{attribute 'GeneratedUsingTerminal: EL1512-0000-0016'}
{attribute addProperty BoxType "EL1512-0000-0016"}
{attribute addProperty Id "Set_counterAT %Q*BOOL1Inhibit_counterAT %Q*BOOL1Set_counter_valueAT %Q*UDINT4"}
{attribute addProperty CRC "2001350844"}
{attribute addProperty Size "6"}
TYPE CNT_Outputs_Channel_774A30BC :
STRUCT
	{attribute addProperty Name "Set_counter"}
	Set_counter AT %Q* : BOOL;
	{attribute addProperty Name "Inhibit_counter"}
	Inhibit_counter AT %Q* : BOOL;
	{attribute addProperty Name "Set_counter_value"}
	Set_counter_value AT %Q* : UDINT;
END_STRUCT
END_TYPE

(* stored: Version 1.2.0.0, ProductVersion 3.1.4024.9
   DUT CNT_Outputs_Channel_774A30BC: Id {11c4018a-45d6-4c90-9c82-aaec7927df72} *)
